{attribute 'GeneratedUsingTerminal: EL6731--0000'}
{attribute addProperty BoxType "EL6731--0000"}
{attribute addProperty Id "InfoDataAT %I*InfoData_90184F0C16"}
{attribute addProperty CRC "554310285"}
{attribute addProperty Size "16"}
TYPE EL6731_210A1A8D EXTENDS EtcSlaveTerminalBase_947E5A46 :
STRUCT
	{attribute addProperty Name "InfoData"}
	InfoData : InfoData_90184F0C;
END_STRUCT
END_TYPE

(* stored: Version 1.2.0.0, ProductVersion 3.1.4024.9
   DUT EL6731_210A1A8D: Id {6e6b16da-0aeb-4ba0-b707-8d1459a70bea} *)
